# EPICS substitutions: iocBoot/iocTml/tml-ch1.substitutions
file "$(TOP)/db/motor.db"
{
    pattern
    { P,                 M,          DESC,          PORT,       ADDR, MRES, ARES, EGU,     DHLM,    DLLM,    VELO, ACCS, TWV  }
    { "SPARC:MOT:TML:", "GUNFLG01", "GUN Flag 1",  "tml-ch1",  0,    1.0,  1.0,  "ustep", 0,  0, 30,   1,    100  }
    { "SPARC:MOT:TML:", "GUNSOLV1", "GUN Sol V1",  "tml-ch1",  1,    1.0,  1.0,  "ustep", 100000,  -100000, 20,   1,    100  }
    { "SPARC:MOT:TML:", "GUNSOLH1", "GUN Sol H1",  "tml-ch1",  2,    1.0,  1.0,  "ustep", 100000,  -100000, 20,   1,    100  }
    { "SPARC:MOT:TML:", "AC1FLG01", "AC1 Flag 1",  "tml-ch1",  3,    1.0,  1.0,  "ustep", 100000,  -100000, 20,   1,    100  }
    { "SPARC:MOT:TML:", "AC2FLG01", "AC2 Flag 1",  "tml-ch1",  4,    1.0,  1.0,  "ustep", 100000,  -100000, 40,   1,    100  }
    { "SPARC:MOT:TML:", "AC3FLG01", "AC3 Flag 1",  "tml-ch1",  5,    1.0,  1.0,  "ustep", 100000,  -100000, 40,   1,    100  }
    { "SPARC:MOT:TML:", "UTLFLG01", "UTL Flag 1",  "tml-ch1",  6,    1.0,  1.0,  "ustep", 100000,  -100000, 40,   1,    100  }
    { "SPARC:MOT:TML:", "UTLFLG02", "UTL Flag 2",  "tml-ch1",  7,    1.0,  1.0,  "ustep", 100000,  -100000, 20,   1,    100  }
    { "SPARC:MOT:TML:", "SBNFLG00", "SBN Flag 0",  "tml-ch1",  8,    1.0,  1.0,  "ustep", 100000,  -100000, 40,   1,    100  }
    { "SPARC:MOT:TML:", "SBNFLG01", "SBN Flag 1",  "tml-ch1",  9,    1.0,  1.0,  "ustep", 100000,  -100000, 40,   1,    100  }
}

#
# Compatibility bridge: provides legacy PV names for the TML OPI screens
# (TML_Main.bob, TML_Control.bob, TML_StatusRegisters.bob, TML_Settings.bob)
#
file "$(TOP)/db/tml_compat.db"
{
    pattern
    { P,                 M,          PORT,       ADDR }
    { "SPARC:MOT:TML:", "GUNFLG01", "tml-ch1",  0    }
    { "SPARC:MOT:TML:", "GUNSOLV1", "tml-ch1",  1    }
    { "SPARC:MOT:TML:", "GUNSOLH1", "tml-ch1",  2    }
    { "SPARC:MOT:TML:", "AC1FLG01", "tml-ch1",  3    }
    { "SPARC:MOT:TML:", "AC2FLG01", "tml-ch1",  4    }
    { "SPARC:MOT:TML:", "AC3FLG01", "tml-ch1",  5    }
    { "SPARC:MOT:TML:", "UTLFLG01", "tml-ch1",  6    }
    { "SPARC:MOT:TML:", "UTLFLG02", "tml-ch1",  7    }
    { "SPARC:MOT:TML:", "SBNFLG00", "tml-ch1",  8    }
    { "SPARC:MOT:TML:", "SBNFLG01", "tml-ch1",  9    }
}
